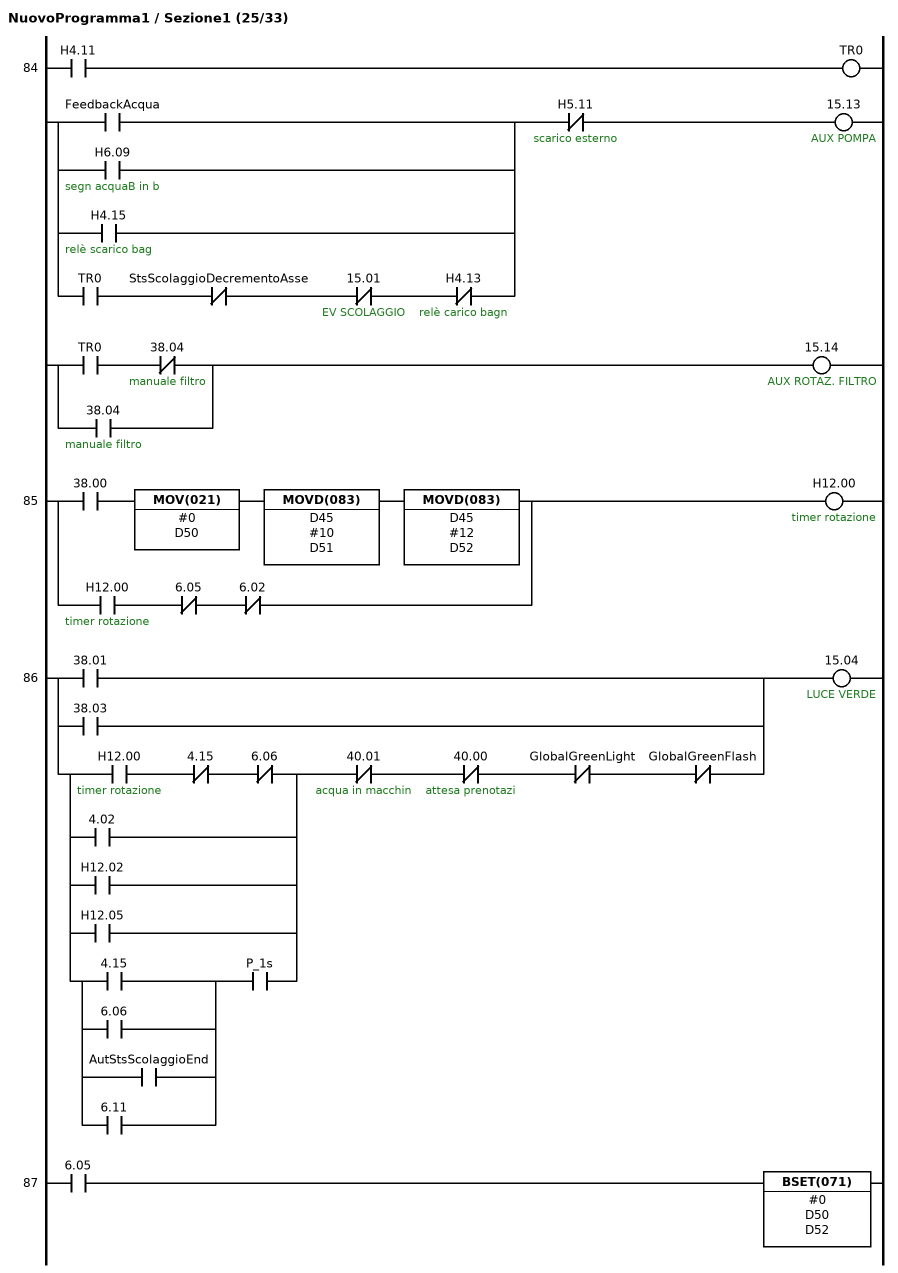
; [picture p24: NuovoProgramma1 / Sezione1, rungs 84-87]
; rung 84
LD FeedbackAcqua
OR H6.09  ; segn acquaB in b
OR H4.15  ; relè scarico bag
LD H4.11
OUT TR0
ANDNOT StsScolaggioDecrementoAsse
ANDNOT 15.01  ; EV SCOLAGGIO
ANDNOT H4.13  ; relè carico bagn
ORLD
ANDNOT H5.11  ; scarico esterno
OUT 15.13  ; AUX POMPA
LD TR0
ANDNOT 38.04  ; manuale filtro
OR 38.04  ; manuale filtro
OUT 15.14  ; AUX ROTAZ. FILTRO
; rung 85
LD 38.00
MOV(021) #0 D50
MOVD(083) D45 #10 D51
MOVD(083) D45 #12 D52
LD H12.00  ; timer rotazione
ANDNOT 6.05
ANDNOT 6.02
ORLD
OUT H12.00  ; timer rotazione
; rung 86
LD 38.01
OR 38.03
LD H12.00  ; timer rotazione
ANDNOT 4.15
ANDNOT 6.06
OR 4.02
OR H12.02
OR H12.05
LD 4.15
OR 6.06
OR AutStsScolaggioEnd
OR 6.11
AND P_1s
ORLD
ANDNOT 40.01  ; acqua in macchin
ANDNOT 40.00  ; attesa prenotazi
ANDNOT GlobalGreenLight
ANDNOT GlobalGreenFlash
ORLD
OUT 15.04  ; LUCE VERDE
; rung 87
LD 6.05
BSET(071) #0 D50 D52

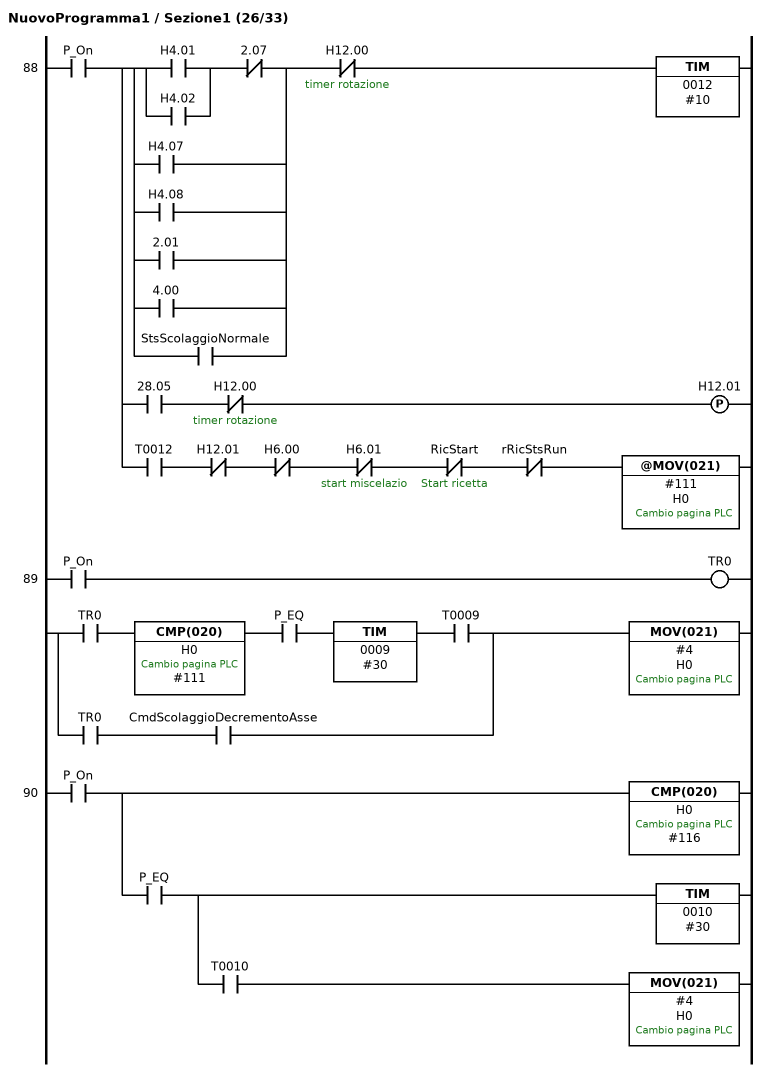
; rung 88
LD P_On
OUT TR0
LD H4.01
OR H4.02
ANDNOT 2.07
OR H4.07
OR H4.08
OR 2.01
OR 4.00
OR StsScolaggioNormale
ANDLD
ANDNOT H12.00  ; timer rotazione
TIM 0012 #10
LD TR0
AND 28.05
ANDNOT H12.00  ; timer rotazione
DIFU(013) H12.01
LD TR0
AND T0012
ANDNOT H12.01
ANDNOT H6.00
ANDNOT H6.01  ; start miscelazio
ANDNOT RicStart  ; Start ricetta
ANDNOT rRicStsRun
@MOV(021) #111 H0  ; Cambio pagina PLC
; rung 89
LD P_On
OUT TR0
CMP(020) H0 #111  ; Cambio pagina PLC
AND P_EQ
TIM 0009 #30
AND T0009
LD TR0
AND CmdScolaggioDecrementoAsse
ORLD
MOV(021) #4 H0  ; Cambio pagina PLC
; rung 90
LD P_On
CMP(020) H0 #116  ; Cambio pagina PLC
AND P_EQ
TIM 0010 #30
AND T0010
MOV(021) #4 H0  ; Cambio pagina PLC

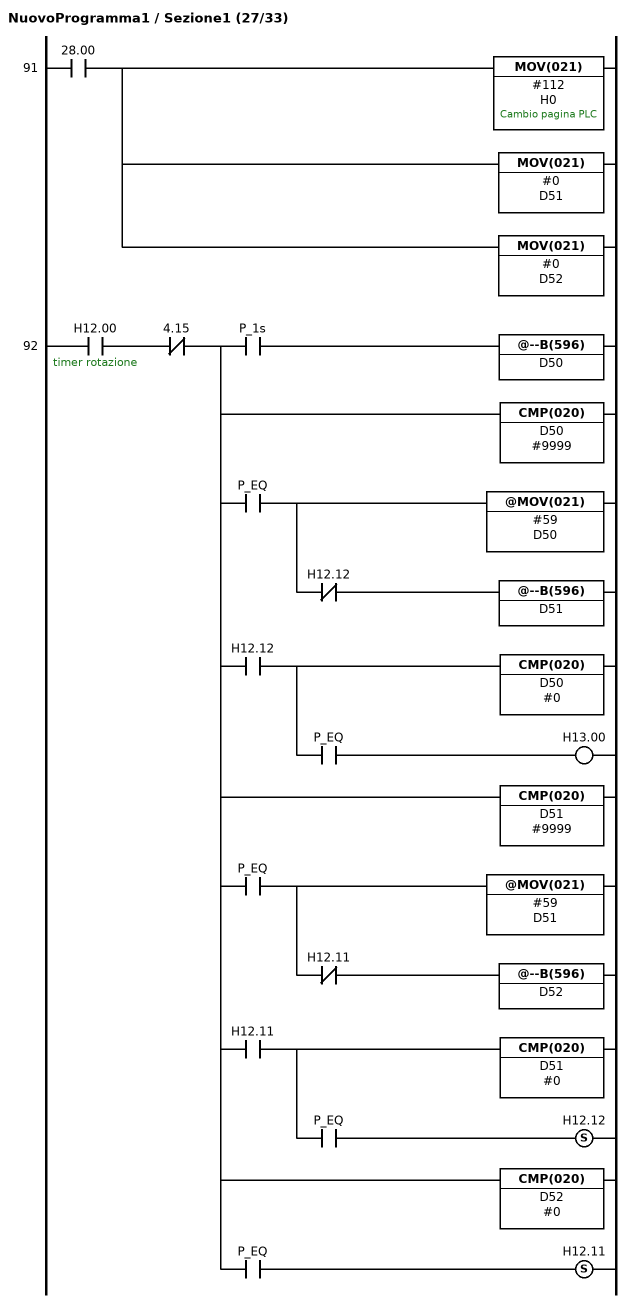
; rung 91
LD 28.00
MOV(021) #112 H0  ; Cambio pagina PLC
MOV(021) #0 D51
MOV(021) #0 D52
; rung 92
LD H12.00  ; timer rotazione
ANDNOT 4.15
OUT TR0
AND P_1s
@--B(596) D50
LD TR0
CMP(020) D50 #9999
AND P_EQ
@MOV(021) #59 D50
ANDNOT H12.12
@--B(596) D51
LD TR0
AND H12.12
CMP(020) D50 #0
AND P_EQ
OUT H13.00
LD TR0
CMP(020) D51 #9999
AND P_EQ
@MOV(021) #59 D51
ANDNOT H12.11
@--B(596) D52
LD TR0
AND H12.11
CMP(020) D51 #0
AND P_EQ
SET H12.12
LD TR0
CMP(020) D52 #0
AND P_EQ
SET H12.11

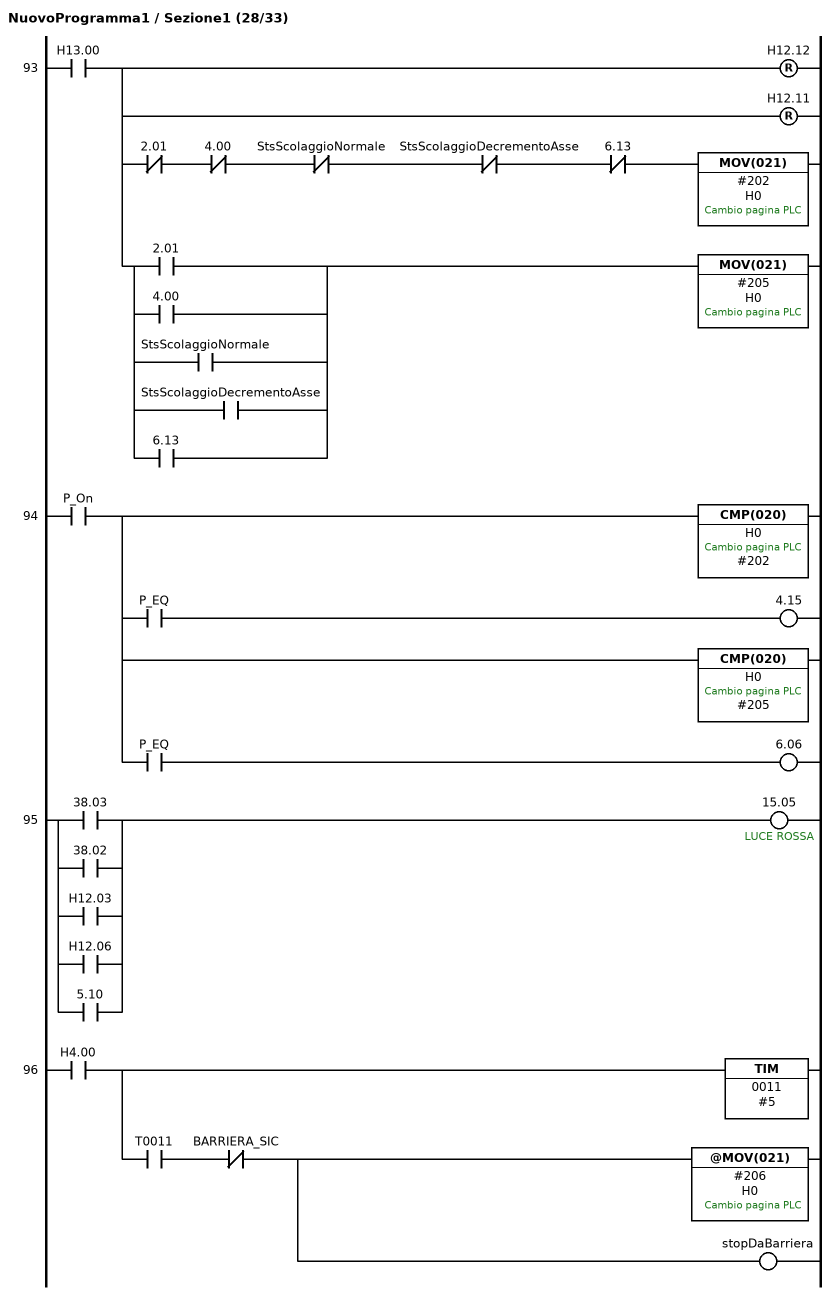
; rung 93
LD H13.00
OUT TR0
RSET H12.12
RSET H12.11
ANDNOT 2.01
ANDNOT 4.00
ANDNOT StsScolaggioNormale
ANDNOT StsScolaggioDecrementoAsse
ANDNOT 6.13
MOV(021) #202 H0  ; Cambio pagina PLC
LD TR0
LD 2.01
OR 4.00
OR StsScolaggioNormale
OR StsScolaggioDecrementoAsse
OR 6.13
ANDLD
MOV(021) #205 H0  ; Cambio pagina PLC
; rung 94
LD P_On
OUT TR0
CMP(020) H0 #202  ; Cambio pagina PLC
AND P_EQ
OUT 4.15
LD TR0
CMP(020) H0 #205  ; Cambio pagina PLC
AND P_EQ
OUT 6.06
; rung 95
LD 38.03
OR 38.02
OR H12.03
OR H12.06
OR 5.10
OUT 15.05  ; LUCE ROSSA
; rung 96
LD H4.00
TIM 0011 #5
AND T0011
ANDNOT BARRIERA_SIC
@MOV(021) #206 H0  ; Cambio pagina PLC
OUT stopDaBarriera

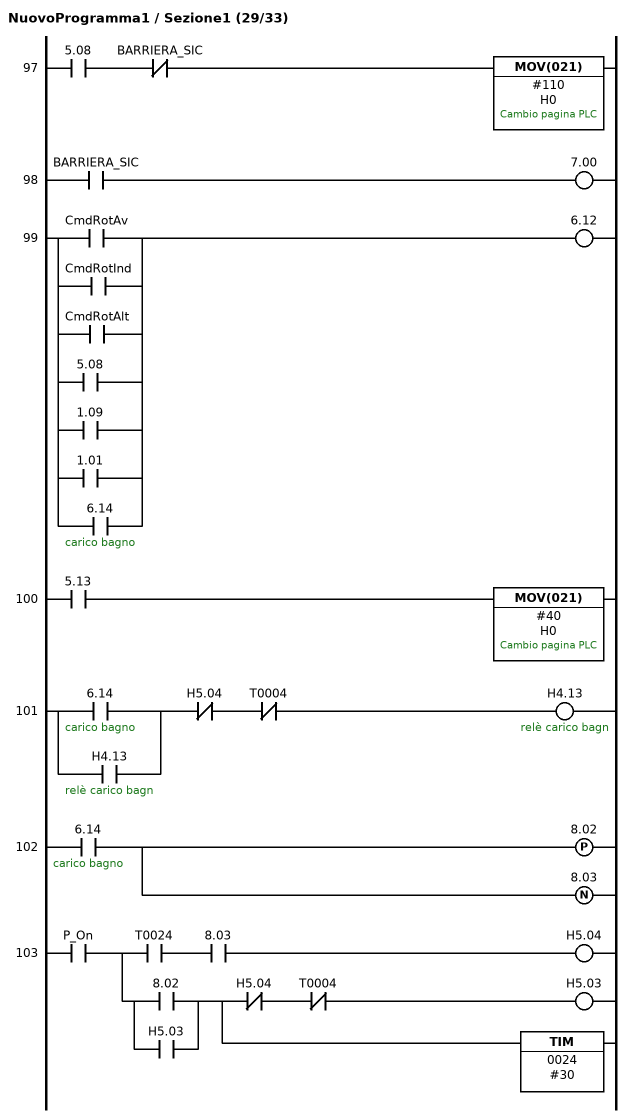
; rung 97
LD 5.08
ANDNOT BARRIERA_SIC
MOV(021) #110 H0  ; Cambio pagina PLC
; rung 98
LD BARRIERA_SIC
OUT 7.00
; rung 99
LD CmdRotAv
OR CmdRotInd
OR CmdRotAlt
OR 5.08
OR 1.09
OR 1.01
OR 6.14  ; carico bagno
OUT 6.12
; rung 100
LD 5.13
MOV(021) #40 H0  ; Cambio pagina PLC
; rung 101
LD 6.14  ; carico bagno
OR H4.13  ; relè carico bagn
ANDNOT H5.04
ANDNOT T0004
OUT H4.13  ; relè carico bagn
; rung 102
LD 6.14  ; carico bagno
DIFU(013) 8.02
DIFD(014) 8.03
; rung 103
LD P_On
OUT TR0
AND T0024
AND 8.03
OUT H5.04
LD TR0
LD 8.02
OR H5.03
ANDLD
OUT TR0
ANDNOT H5.04
ANDNOT T0004
OUT H5.03
LD TR0
TIM 0024 #30

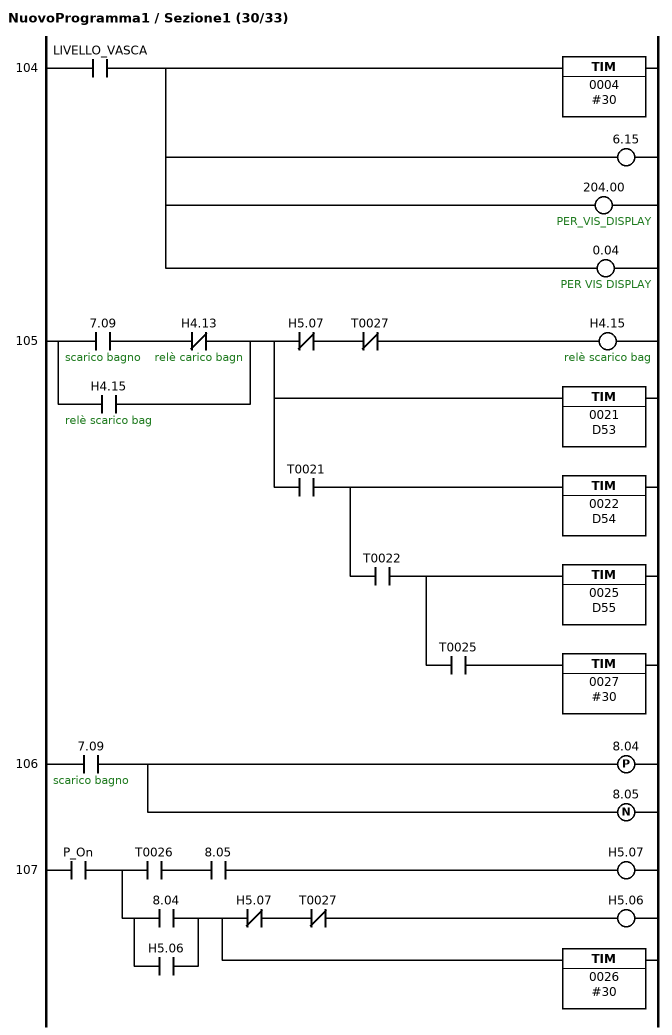
; rung 104
LD LIVELLO_VASCA
TIM 0004 #30
OUT 6.15
OUT 204.00  ; PER_VIS_DISPLAY
OUT 0.04  ; PER VIS DISPLAY
; rung 105
LD 7.09  ; scarico bagno
ANDNOT H4.13  ; relè carico bagn
OR H4.15  ; relè scarico bag
OUT TR0
ANDNOT H5.07
ANDNOT T0027
OUT H4.15  ; relè scarico bag
LD TR0
TIM 0021 D53
AND T0021
TIM 0022 D54
AND T0022
TIM 0025 D55
AND T0025
TIM 0027 #30
; rung 106
LD 7.09  ; scarico bagno
DIFU(013) 8.04
DIFD(014) 8.05
; rung 107
LD P_On
OUT TR0
AND T0026
AND 8.05
OUT H5.07
LD TR0
LD 8.04
OR H5.06
ANDLD
OUT TR0
ANDNOT H5.07
ANDNOT T0027
OUT H5.06
LD TR0
TIM 0026 #30

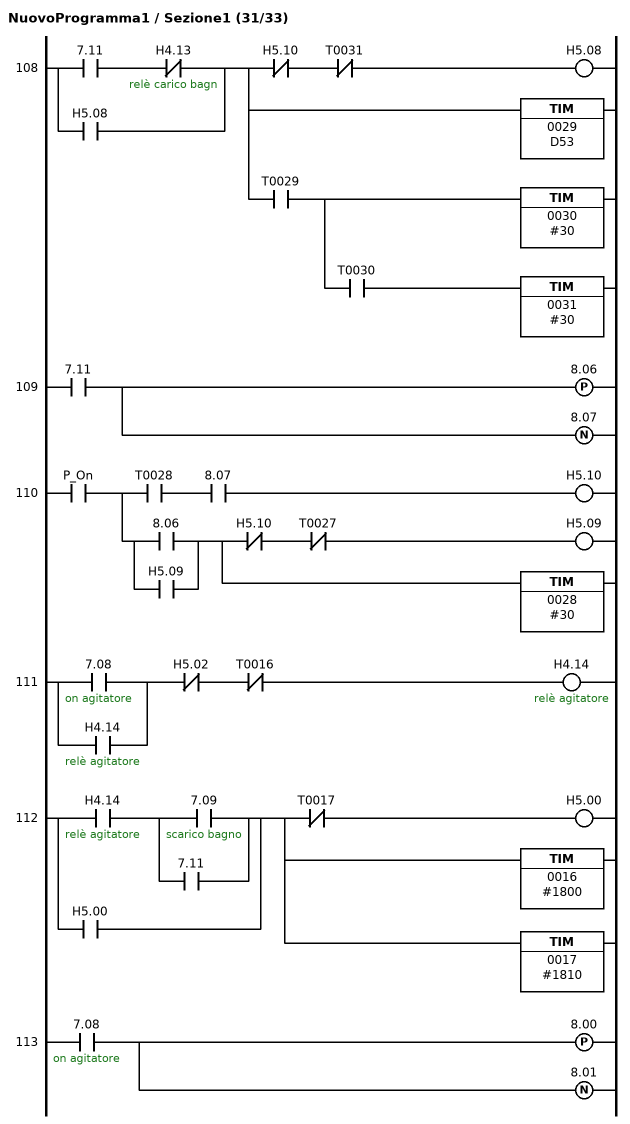
; rung 108
LD 7.11
ANDNOT H4.13  ; relè carico bagn
OR H5.08
OUT TR0
ANDNOT H5.10
ANDNOT T0031
OUT H5.08
LD TR0
TIM 0029 D53
AND T0029
TIM 0030 #30
AND T0030
TIM 0031 #30
; rung 109
LD 7.11
DIFU(013) 8.06
DIFD(014) 8.07
; rung 110
LD P_On
OUT TR0
AND T0028
AND 8.07
OUT H5.10
LD TR0
LD 8.06
OR H5.09
ANDLD
OUT TR0
ANDNOT H5.10
ANDNOT T0027
OUT H5.09
LD TR0
TIM 0028 #30
; rung 111
LD 7.08  ; on agitatore
OR H4.14  ; relè agitatore
ANDNOT H5.02
ANDNOT T0016
OUT H4.14  ; relè agitatore
; rung 112
LD H4.14  ; relè agitatore
LD 7.09  ; scarico bagno
OR 7.11
ANDLD
OR H5.00
OUT TR0
ANDNOT T0017
OUT H5.00
LD TR0
TIM 0016 #1800
TIM 0017 #1810
; rung 113
LD 7.08  ; on agitatore
DIFU(013) 8.00
DIFD(014) 8.01

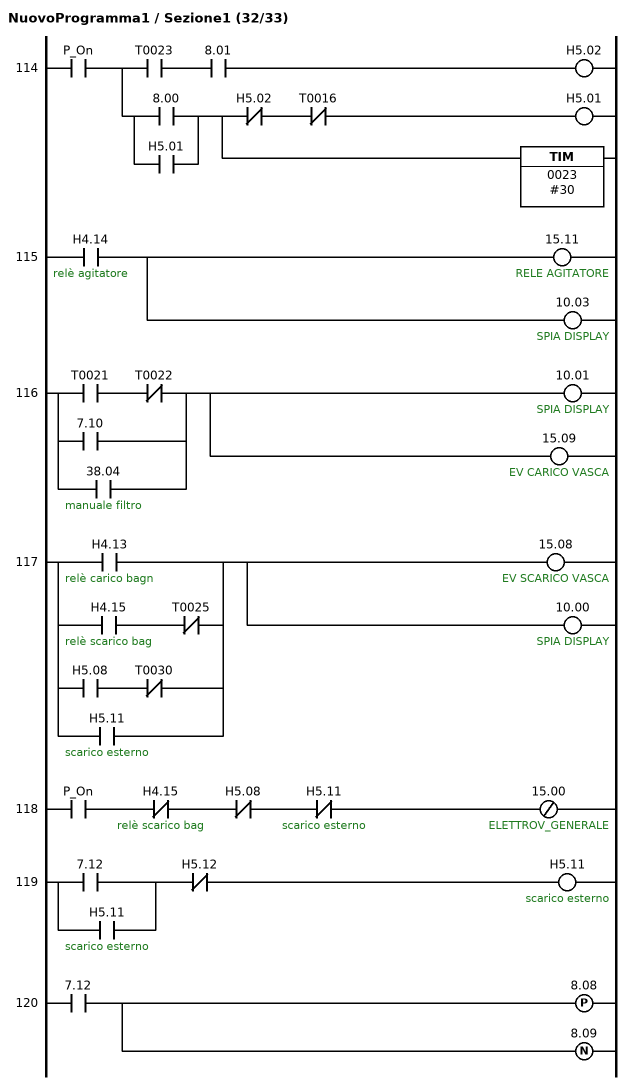
; rung 114
LD P_On
OUT TR0
AND T0023
AND 8.01
OUT H5.02
LD TR0
LD 8.00
OR H5.01
ANDLD
OUT TR0
ANDNOT H5.02
ANDNOT T0016
OUT H5.01
LD TR0
TIM 0023 #30
; rung 115
LD H4.14  ; relè agitatore
OUT 15.11  ; RELE AGITATORE
OUT 10.03  ; SPIA DISPLAY
; rung 116
LD T0021
ANDNOT T0022
OR 7.10
OR 38.04  ; manuale filtro
OUT 10.01  ; SPIA DISPLAY
OUT 15.09  ; EV CARICO VASCA
; rung 117
LD H4.13  ; relè carico bagn
LD H4.15  ; relè scarico bag
ANDNOT T0025
ORLD
LD H5.08
ANDNOT T0030
ORLD
OR H5.11  ; scarico esterno
OUT 15.08  ; EV SCARICO VASCA
OUT 10.00  ; SPIA DISPLAY
; rung 118
LD P_On
ANDNOT H4.15  ; relè scarico bag
ANDNOT H5.08
ANDNOT H5.11  ; scarico esterno
OUTNOT 15.00  ; ELETTROV_GENERALE
; rung 119
LD 7.12
OR H5.11  ; scarico esterno
ANDNOT H5.12
OUT H5.11  ; scarico esterno
; rung 120
LD 7.12
DIFU(013) 8.08
DIFD(014) 8.09

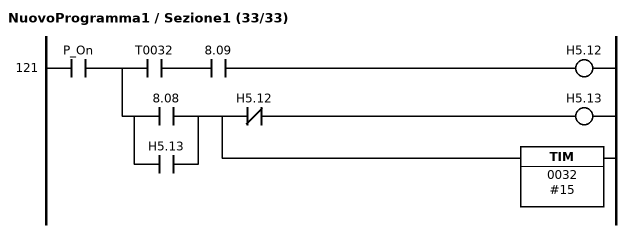
; rung 121
LD P_On
OUT TR0
AND T0032
AND 8.09
OUT H5.12
LD TR0
LD 8.08
OR H5.13
ANDLD
OUT TR0
ANDNOT H5.12
OUT H5.13
LD TR0
TIM 0032 #15

### Section Sezione2

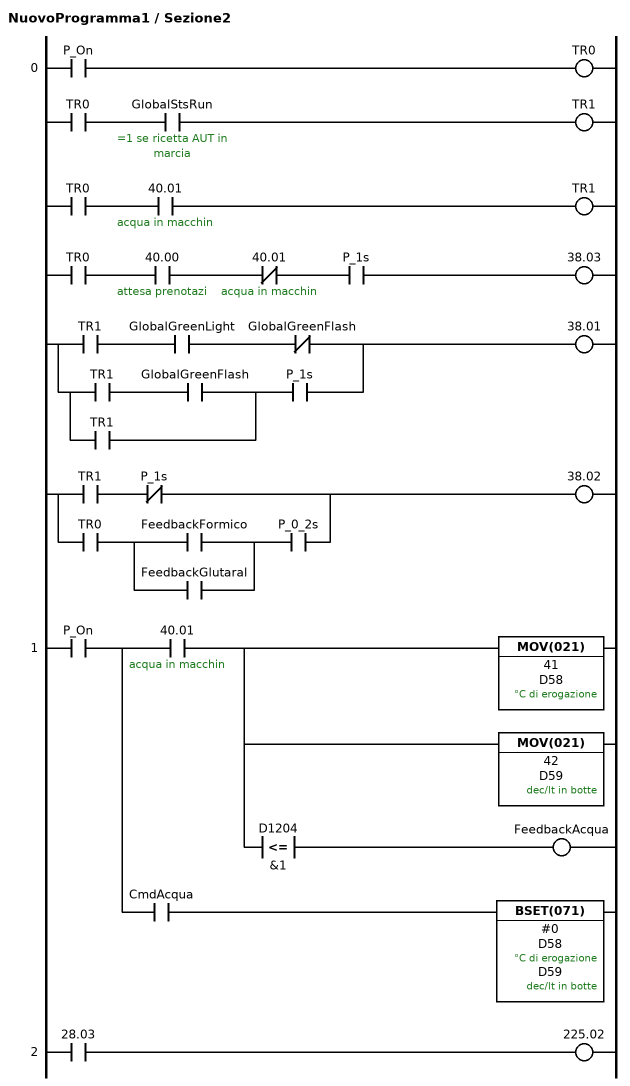
; rung 0
LD P_On
OUT TR0
AND 40.00  ; attesa prenotazi
ANDNOT 40.01  ; acqua in macchin
AND P_1s
OUT 38.03
LD TR0
AND GlobalStsRun  ; =1 se ricetta AUT in marcia
OUT TR1
AND GlobalGreenLight
ANDNOT GlobalGreenFlash
LD TR1
AND GlobalGreenFlash
LD TR0
AND 40.01  ; acqua in macchin
OUT TR1
ORLD
AND P_1s
ORLD
OUT 38.01
LD TR1
ANDNOT P_1s
LD TR0
LD FeedbackFormico
OR FeedbackGlutaral
ANDLD
AND P_0_2s
ORLD
OUT 38.02
; rung 1
LD P_On
OUT TR0
AND 40.01  ; acqua in macchin
MOV(021) 41 D58  ; °C di erogazione
MOV(021) 42 D59  ; dec/lt in botte
AND<=(315) D1204 &1
OUT FeedbackAcqua
LD TR0
AND CmdAcqua
BSET(071) #0 D58 D59  ; °C di erogazione, dec/lt in botte
; rung 2
LD 28.03
OUT 225.02

### Section Sezione3

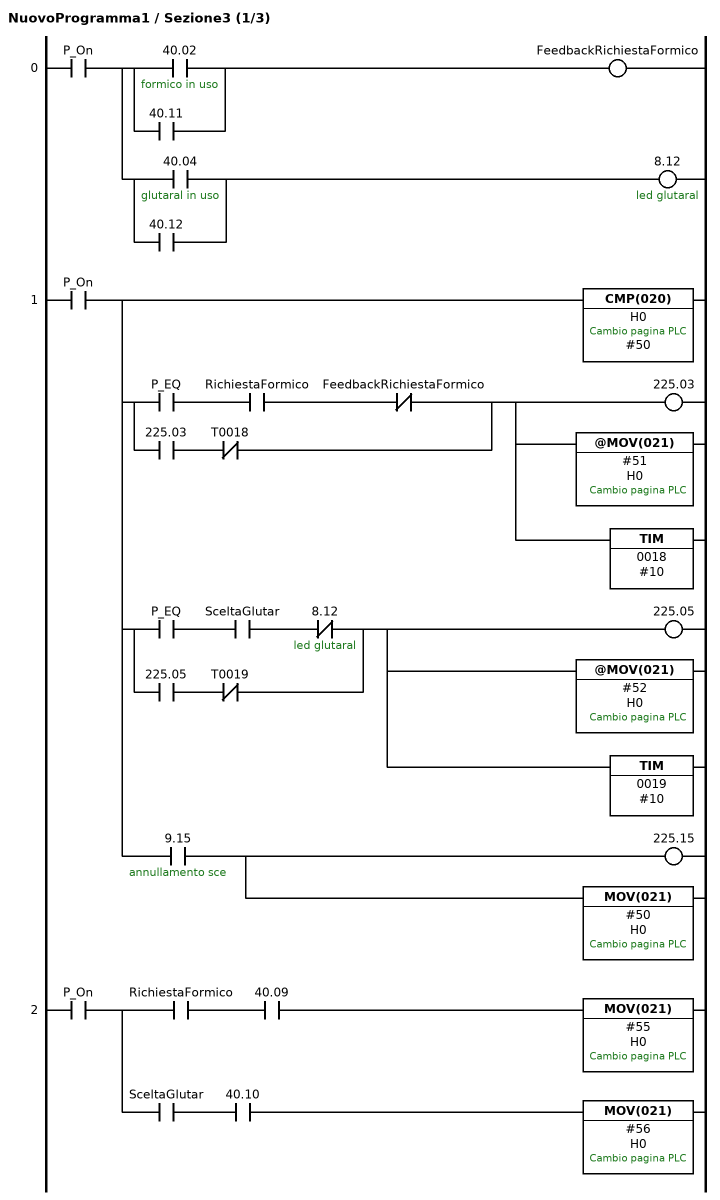
; rung 0
LD P_On
OUT TR0
LD 40.02  ; formico in uso
OR 40.11
ANDLD
OUT FeedbackRichiestaFormico
LD TR0
LD 40.04  ; glutaral in uso
OR 40.12
ANDLD
OUT 8.12  ; led glutaral
; rung 1
LD P_On
OUT TR0
CMP(020) H0 #50  ; Cambio pagina PLC
LD P_EQ
AND RichiestaFormico
ANDNOT FeedbackRichiestaFormico
LD 225.03
ANDNOT T0018
ORLD
ANDLD
OUT 225.03
@MOV(021) #51 H0  ; Cambio pagina PLC
TIM 0018 #10
LD TR0
LD P_EQ
AND SceltaGlutar
ANDNOT 8.12  ; led glutaral
LD 225.05
ANDNOT T0019
ORLD
ANDLD
OUT 225.05
@MOV(021) #52 H0  ; Cambio pagina PLC
TIM 0019 #10
LD TR0
AND 9.15  ; annullamento sce
OUT 225.15
MOV(021) #50 H0  ; Cambio pagina PLC
; rung 2
LD P_On
OUT TR0
AND RichiestaFormico
AND 40.09
MOV(021) #55 H0  ; Cambio pagina PLC
LD TR0
AND SceltaGlutar
AND 40.10
MOV(021) #56 H0  ; Cambio pagina PLC

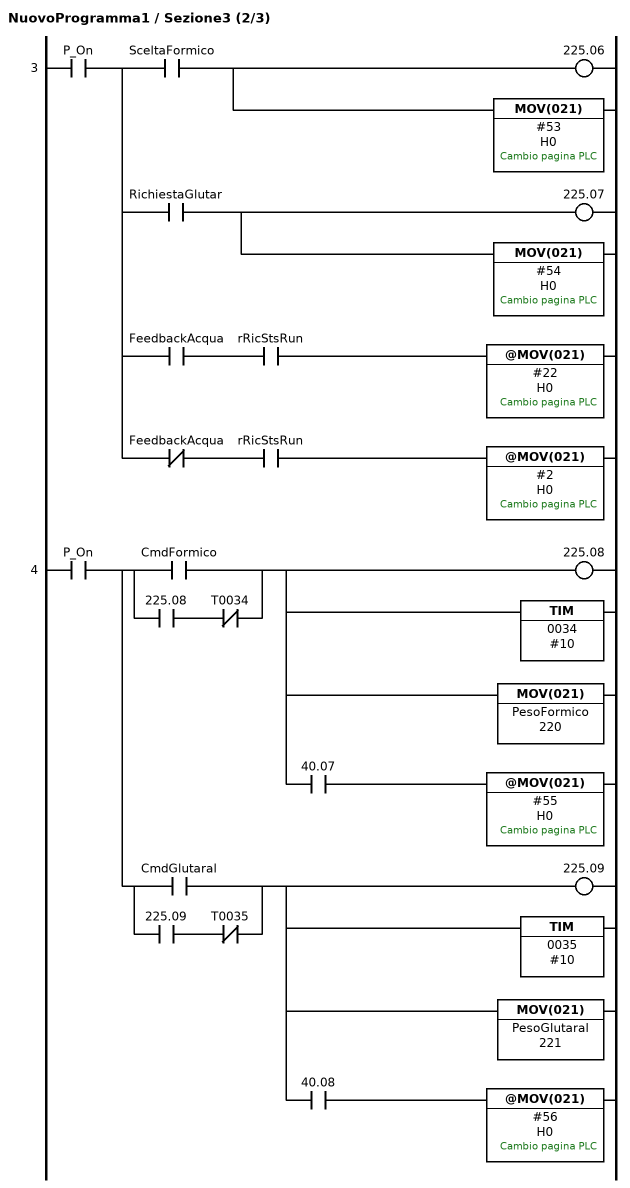
; rung 3
LD P_On
OUT TR0
AND SceltaFormico
OUT 225.06
MOV(021) #53 H0  ; Cambio pagina PLC
LD TR0
AND RichiestaGlutar
OUT 225.07
MOV(021) #54 H0  ; Cambio pagina PLC
LD TR0
AND FeedbackAcqua
AND rRicStsRun
@MOV(021) #22 H0  ; Cambio pagina PLC
LD TR0
ANDNOT FeedbackAcqua
AND rRicStsRun
@MOV(021) #2 H0  ; Cambio pagina PLC
; rung 4
LD P_On
OUT TR0
LD CmdFormico
LD 225.08
ANDNOT T0034
ORLD
ANDLD
OUT 225.08
TIM 0034 #10
MOV(021) PesoFormico 220
AND 40.07
@MOV(021) #55 H0  ; Cambio pagina PLC
LD TR0
LD CmdGlutaral
LD 225.09
ANDNOT T0035
ORLD
ANDLD
OUT 225.09
TIM 0035 #10
MOV(021) PesoGlutaral 221
AND 40.08
@MOV(021) #56 H0  ; Cambio pagina PLC

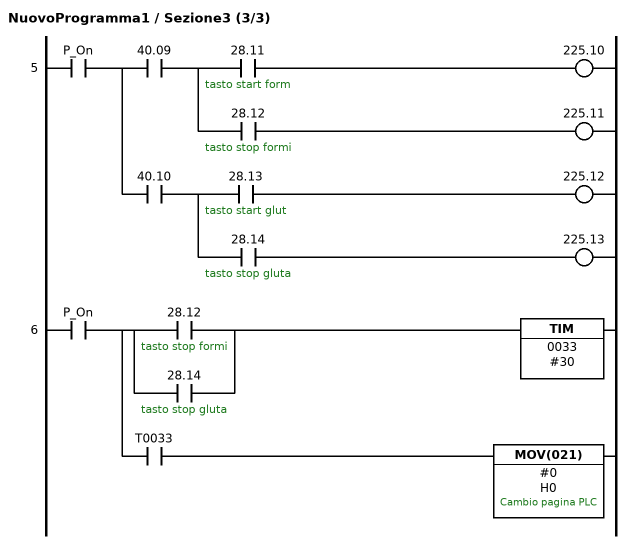
; rung 5
LD P_On
OUT TR0
AND 40.09
OUT TR1
AND 28.11  ; tasto start form
OUT 225.10
LD TR1
AND 28.12  ; tasto stop formi
OUT 225.11
LD TR0
AND 40.10
OUT TR0
AND 28.13  ; tasto start glut
OUT 225.12
LD TR0
AND 28.14  ; tasto stop gluta
OUT 225.13
; rung 6
LD P_On
OUT TR0
LD 28.12  ; tasto stop formi
OR 28.14  ; tasto stop gluta
ANDLD
TIM 0033 #30
LD TR0
AND T0033
MOV(021) #0 H0  ; Cambio pagina PLC
; rung 7
END(001)

## Program TaskRicette (cyclic task 1)

### Section CambioPagina

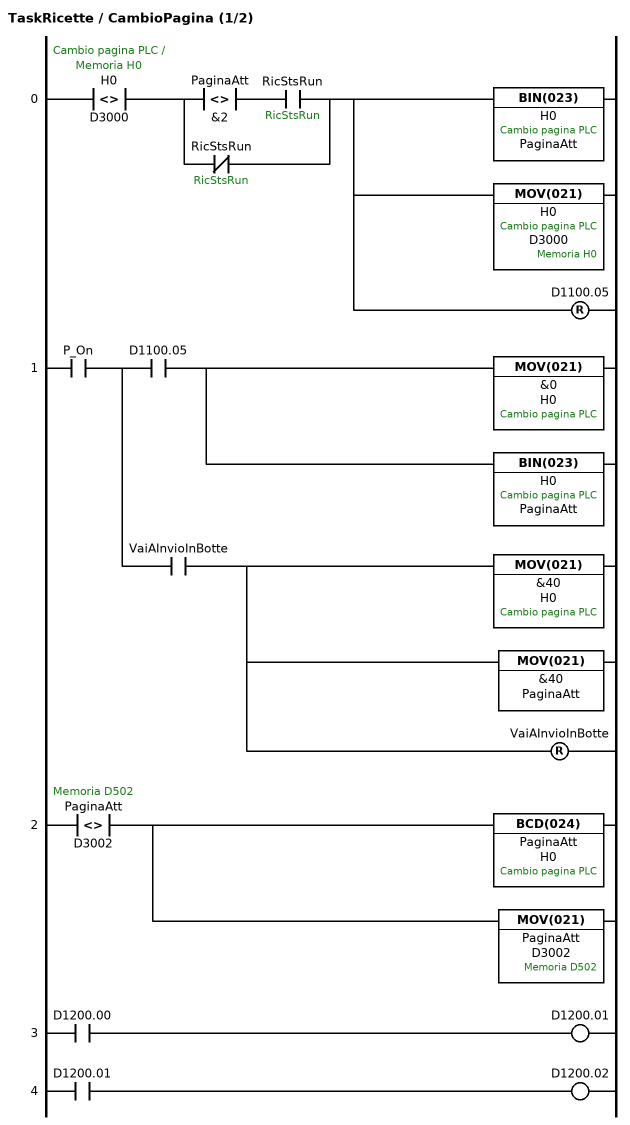
; rung 0
LD<>(305) H0 D3000  ; Cambio pagina PLC, Memoria H0
LD<>(305) PaginaAtt &2
AND RicStsRun  ; RicStsRun
ORNOT RicStsRun  ; RicStsRun
ANDLD
BIN(023) H0 PaginaAtt  ; Cambio pagina PLC
MOV(021) H0 D3000  ; Cambio pagina PLC, Memoria H0
RSET D1100.05
; rung 1
LD P_On
OUT TR0
AND D1100.05
MOV(021) &0 H0  ; Cambio pagina PLC
BIN(023) H0 PaginaAtt  ; Cambio pagina PLC
LD TR0
AND VaiAInvioInBotte
MOV(021) &40 H0  ; Cambio pagina PLC
MOV(021) &40 PaginaAtt
RSET VaiAInvioInBotte
; rung 2
LD<>(305) PaginaAtt D3002  ; Memoria D502
BCD(024) PaginaAtt H0  ; Cambio pagina PLC
MOV(021) PaginaAtt D3002  ; Memoria D502
; rung 3
LD D1200.00
OUT D1200.01
; rung 4
LD D1200.01
OUT D1200.02

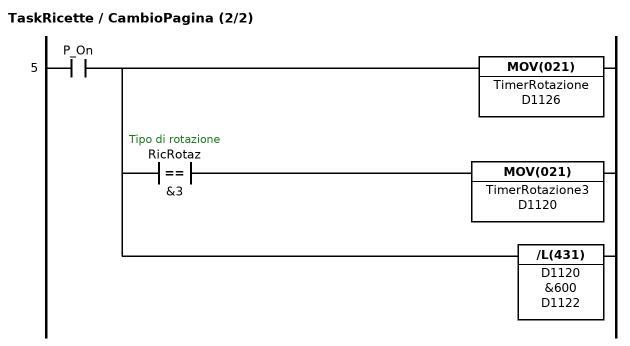
; rung 5
LD P_On
OUT TR0
MOV(021) TimerRotazione D1126
AND=(300) RicRotaz &3  ; Tipo di rotazione
MOV(021) TimerRotazione3 D1120
LD TR0
/L(431) D1120 &600 D1122

### Section Puntatori

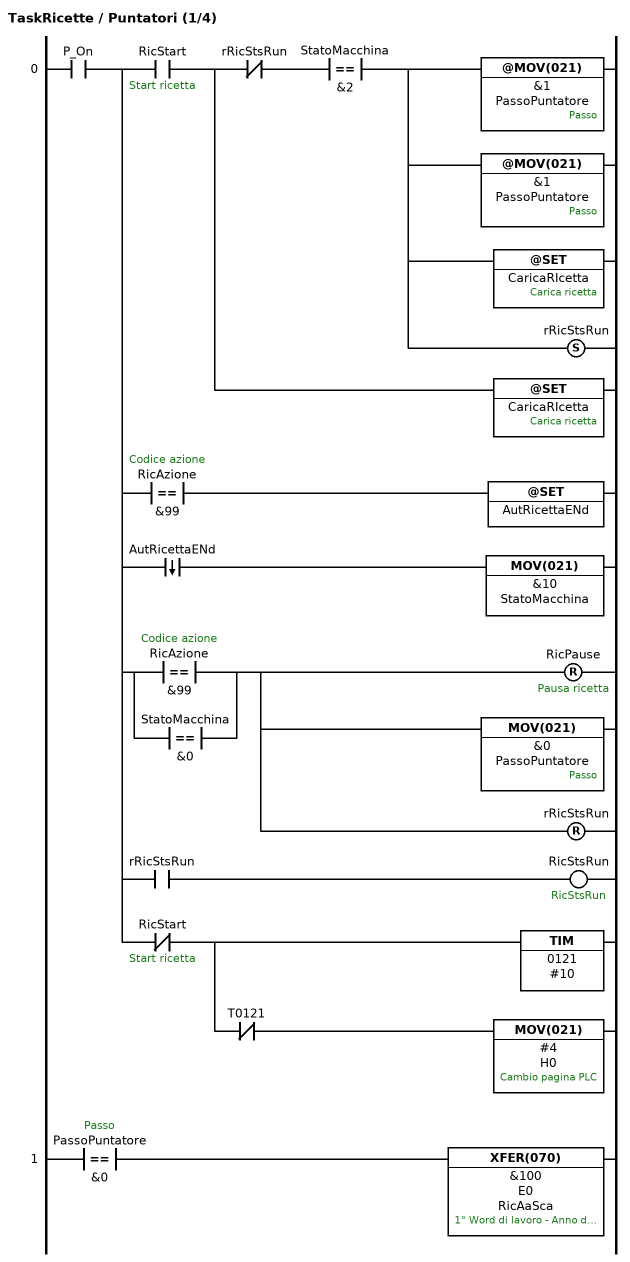
; rung 0
LD P_On
OUT TR0
AND RicStart  ; Start ricetta
OUT TR1
ANDNOT rRicStsRun
AND=(300) StatoMacchina &2
@MOV(021) &1 PassoPuntatore  ; Passo
@MOV(021) &1 PassoPuntatore  ; Passo
@SET CaricaRIcetta  ; Carica ricetta
SET rRicStsRun
LD TR1
@SET CaricaRIcetta  ; Carica ricetta
LD TR0
AND=(300) RicAzione &99  ; Codice azione
@SET AutRicettaENd
LD TR0
%AND AutRicettaENd
MOV(021) &10 StatoMacchina
LD TR0
LD=(300) RicAzione &99  ; Codice azione
OR=(300) StatoMacchina &0
ANDLD
RSET RicPause  ; Pausa ricetta
MOV(021) &0 PassoPuntatore  ; Passo
RSET rRicStsRun
LD TR0
AND rRicStsRun
OUT RicStsRun  ; RicStsRun
LD TR0
ANDNOT RicStart  ; Start ricetta
TIM 0121 #10
ANDNOT T0121
MOV(021) #4 H0  ; Cambio pagina PLC
; rung 1
LD=(300) PassoPuntatore &0  ; Passo
XFER(070) &100 E0 RicAaSca  ; 1° Word di lavoro - Anno di produzione

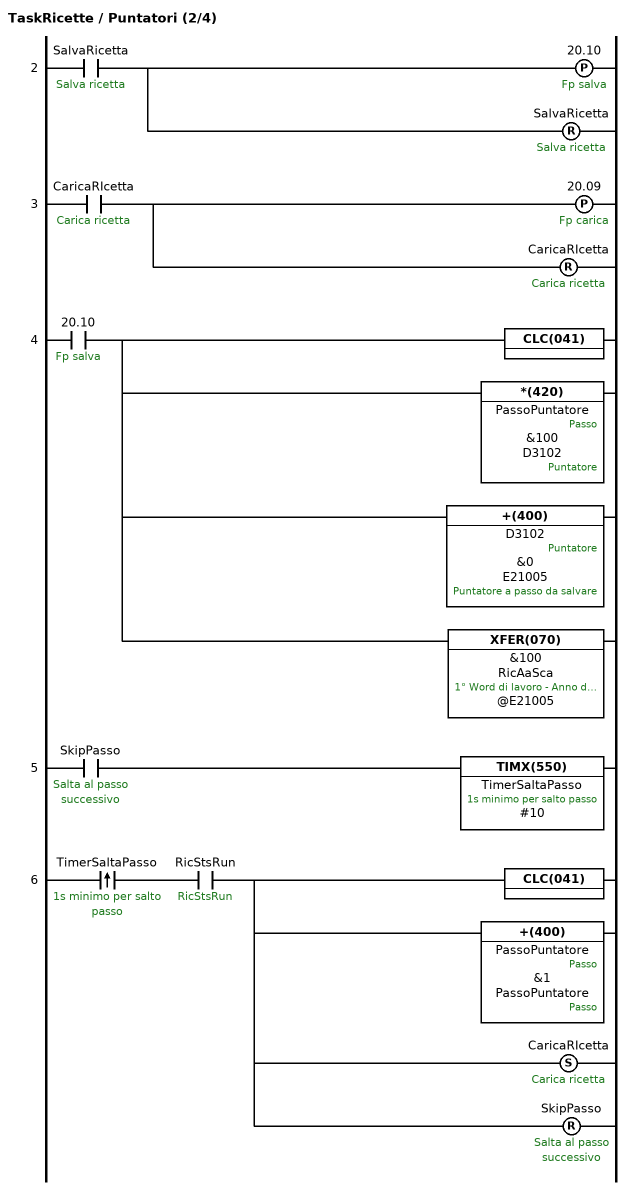
; rung 2
LD SalvaRicetta  ; Salva ricetta
DIFU(013) 20.10  ; Fp salva
RSET SalvaRicetta  ; Salva ricetta
; rung 3
LD CaricaRIcetta  ; Carica ricetta
DIFU(013) 20.09  ; Fp carica
RSET CaricaRIcetta  ; Carica ricetta
; rung 4
LD 20.10  ; Fp salva
CLC(041)
*(420) PassoPuntatore &100 D3102  ; Passo, Puntatore
+(400) D3102 &0 E21005  ; Puntatore, Puntatore a passo da salvare
XFER(070) &100 RicAaSca @E21005  ; 1° Word di lavoro - Anno di produzione
; rung 5
LD SkipPasso  ; Salta al passo successivo
TIMX(550) TimerSaltaPasso #10  ; 1s minimo per salto passo
; rung 6
@LD TimerSaltaPasso  ; 1s minimo per salto passo
AND RicStsRun  ; RicStsRun
CLC(041)
+(400) PassoPuntatore &1 PassoPuntatore  ; Passo
SET CaricaRIcetta  ; Carica ricetta
RSET SkipPasso  ; Salta al passo successivo

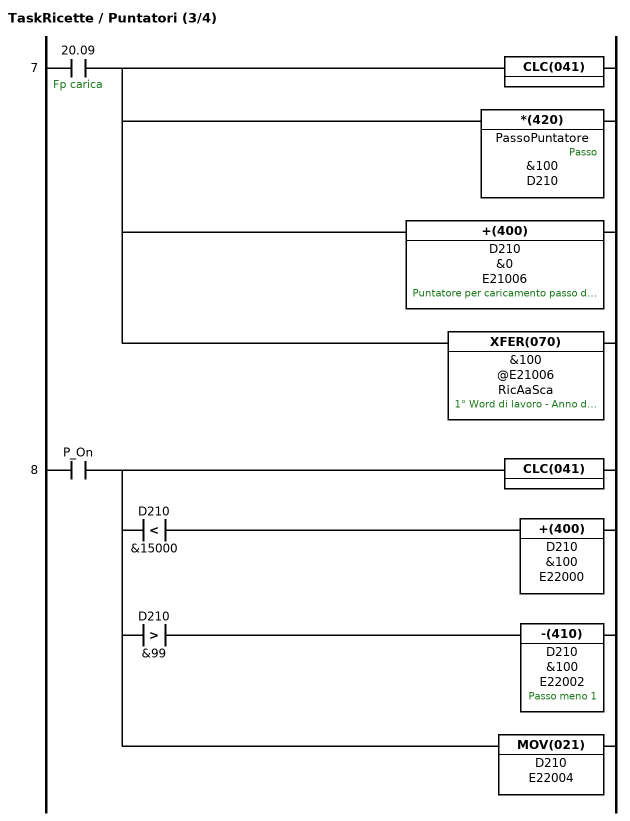
; rung 7
LD 20.09  ; Fp carica
CLC(041)
*(420) PassoPuntatore &100 D210  ; Passo
+(400) D210 &0 E21006  ; Puntatore per caricamento passo da DB a lavoro
XFER(070) &100 @E21006 RicAaSca  ; 1° Word di lavoro - Anno di produzione
; rung 8
LD P_On
OUT TR0
CLC(041)
AND<(310) D210 &15000
+(400) D210 &100 E22000
LD TR0
AND>(320) D210 &99
-(410) D210 &100 E22002  ; Passo meno 1
LD TR0
MOV(021) D210 E22004

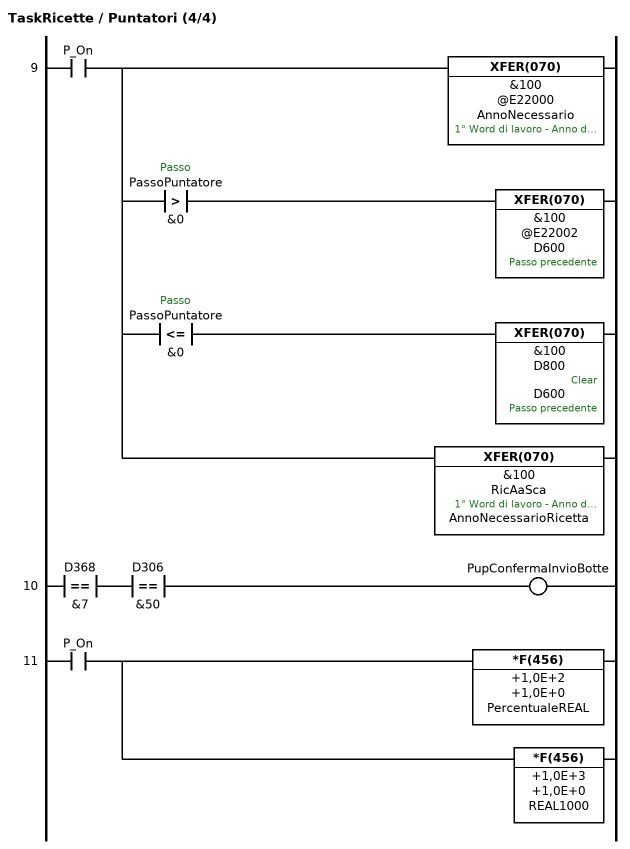
; rung 9
LD P_On
OUT TR0
XFER(070) &100 @E22000 AnnoNecessario  ; 1° Word di lavoro - Anno di produzione
AND>(320) PassoPuntatore &0  ; Passo
XFER(070) &100 @E22002 D600  ; Passo precedente
LD TR0
AND<=(315) PassoPuntatore &0  ; Passo
XFER(070) &100 D800 D600  ; Clear, Passo precedente
LD TR0
XFER(070) &100 RicAaSca AnnoNecessarioRicetta  ; 1° Word di lavoro - Anno di produzione
; rung 10
LD=(300) D368 &7
AND=(300) D306 &50
OUT PupConfermaInvioBotte
; rung 11
LD P_On
*F(456) +1,0E+2 +1,0E+0 PercentualeREAL
*F(456) +1,0E+3 +1,0E+0 REAL1000

### Section StatoRicetta

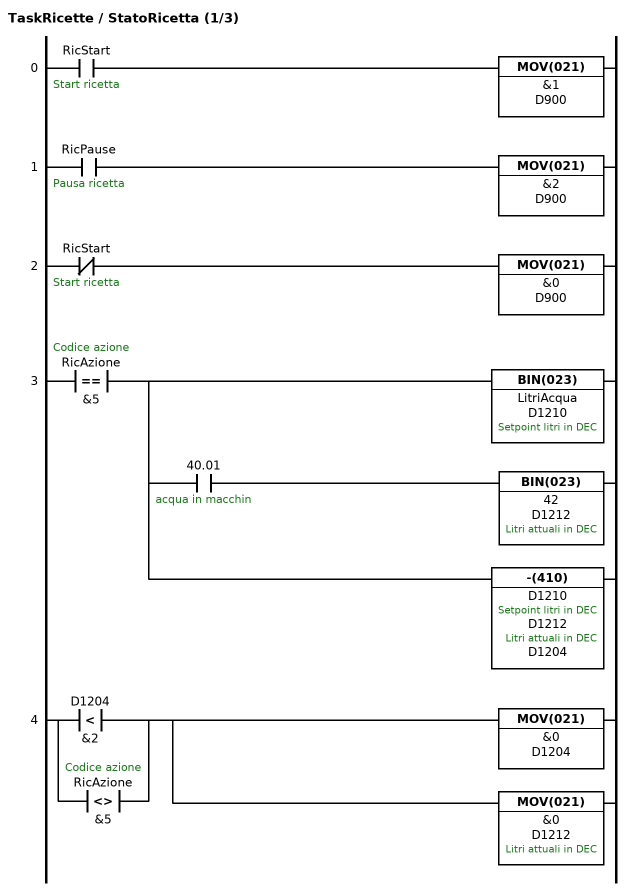
; rung 0
LD RicStart  ; Start ricetta
MOV(021) &1 D900
; rung 1
LD RicPause  ; Pausa ricetta
MOV(021) &2 D900
; rung 2
LDNOT RicStart  ; Start ricetta
MOV(021) &0 D900
; rung 3
LD=(300) RicAzione &5  ; Codice azione
OUT TR0
BIN(023) LitriAcqua D1210  ; Setpoint litri in DEC
AND 40.01  ; acqua in macchin
BIN(023) 42 D1212  ; Litri attuali in DEC
LD TR0
-(410) D1210 D1212 D1204  ; Setpoint litri in DEC, Litri attuali in DEC
; rung 4
LD<(310) D1204 &2
OR<>(305) RicAzione &5  ; Codice azione
MOV(021) &0 D1204
MOV(021) &0 D1212  ; Litri attuali in DEC

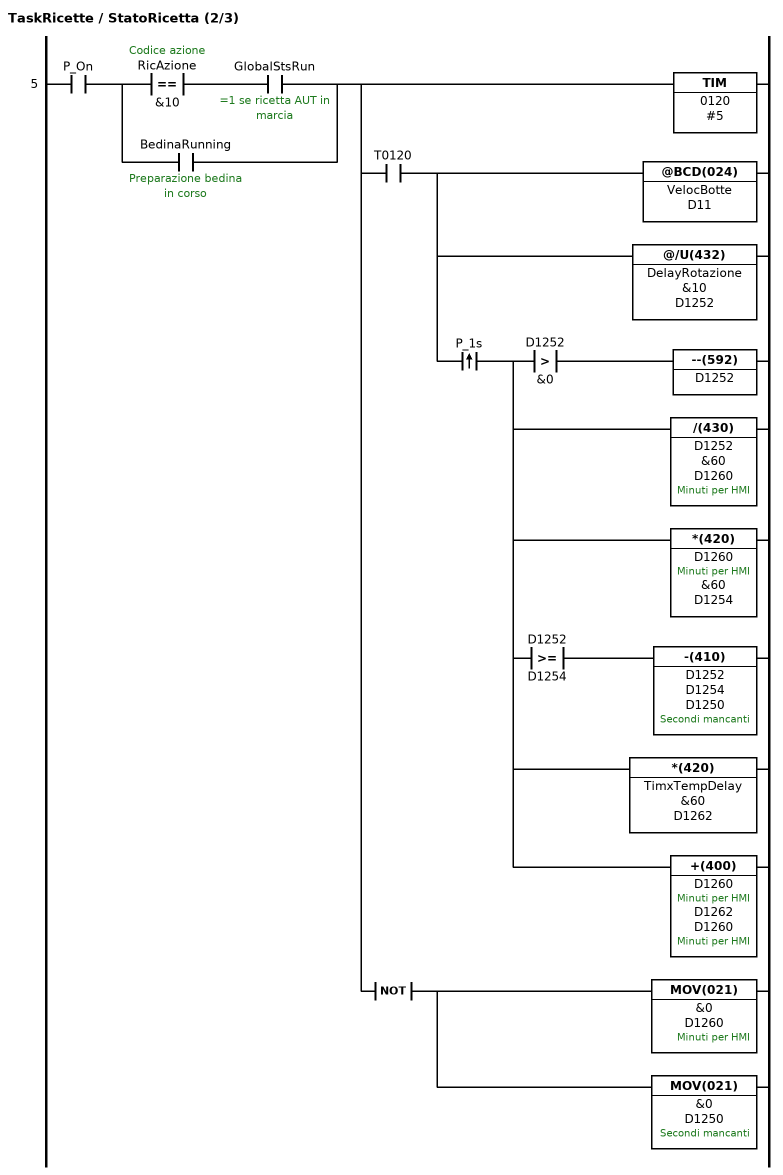
; rung 5
LD P_On
LD=(300) RicAzione &10  ; Codice azione
AND GlobalStsRun  ; =1 se ricetta AUT in marcia
OR BedinaRunning  ; Preparazione bedina in corso
ANDLD
OUT TR0
TIM 0120 #5
AND T0120
@BCD(024) VelocBotte D11
@/U(432) DelayRotazione &10 D1252
@AND P_1s
OUT TR1
AND>(320) D1252 &0
--(592) D1252
LD TR1
/(430) D1252 &60 D1260  ; Minuti per HMI
*(420) D1260 &60 D1254  ; Minuti per HMI
AND>=(325) D1252 D1254
-(410) D1252 D1254 D1250  ; Secondi mancanti
LD TR1
*(420) TimxTempDelay &60 D1262
+(400) D1260 D1262 D1260  ; Minuti per HMI
LD TR0
NOT(520)
MOV(021) &0 D1260  ; Minuti per HMI
MOV(021) &0 D1250  ; Secondi mancanti

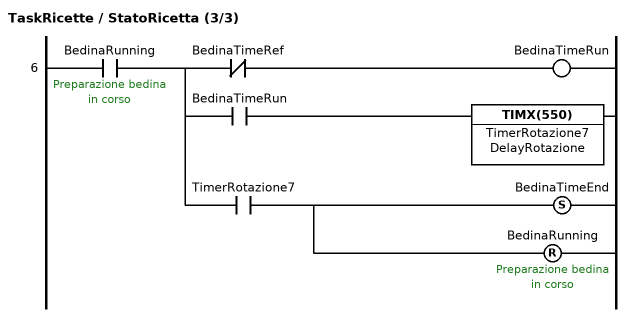
; rung 6
LD BedinaRunning  ; Preparazione bedina in corso
OUT TR0
ANDNOT BedinaTimeRef
OUT BedinaTimeRun
LD TR0
AND BedinaTimeRun
TIMX(550) TimerRotazione7 DelayRotazione
LD TR0
AND TimerRotazione7
SET BedinaTimeEnd
RSET BedinaRunning  ; Preparazione bedina in corso

### Section END

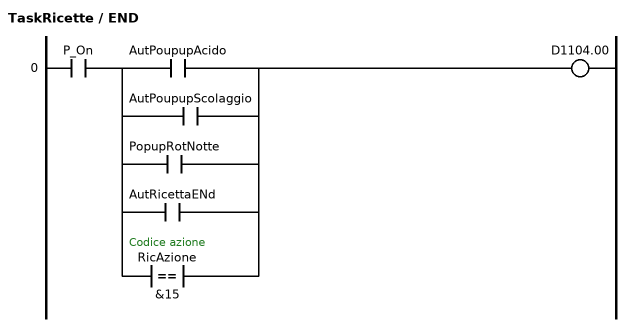
; rung 0
LD P_On
LD AutPoupupAcido
OR AutPoupupScolaggio
OR PopupRotNotte
OR AutRicettaENd
OR=(300) RicAzione &15  ; Codice azione
ANDLD
OUT D1104.00
; rung 1
END(001)

## Program CicliStep (cyclic task 2)
Local symbols
CmdRst D2000.00 BOOL
CmdStart D2000.01 BOOL
Index D2010 INT
MemRiga D2012 WORD
StepCiclo D2001.00 BOOL[15]
StsEnd D2000.02 BOOL
StsRun D2000.03 BOOL
TempAnnoNecessario D2016 DINT
i D2014 INT
 IF TimerSaltaPasso.CF = TRUE  AND MemTimSkip=FALSE THEN
	Index:= 1;
	CmdRotAv:= false;
	CmdRotInd:= false;
	CmdRotAlt:= false;
	CmdRotStop:= false;
	CmdRotNotte:= false;
	CmdAcqua:= false;
	CmdFormico:= false;
	CmdGlutaral:= false;
	CmdScolaggioDecrementoAsse:= false;
	CmdScolaggioNormale:= false;
	PopupMancatoScolaggio:= false;
	RichiestaLetturaBarcode:= false;
	AutCmdNotturno:= false;
	AutPoupupScolaggio:= false;

end_if;
MemTimSkip:= TimerSaltaPasso.CF;
 
 (*Stop Riga*)
IF NOT  RicStart then
	StsRun:= false;
	StsEnd:= true;
	Index:= 5;
END_IF;
 
 
 (* Reset ciclo e comandi vari *)
IF CmdRst = TRUE THEN
	StsRun:= false;
	CmdStart:= false;
	CmdRst := false;	
END_IF;
GlobalGreenFlash:= false;
GlobalGreenLight:= false;
LetturaPesoREAL:= DINT_TO_REAL(LetturaPesoDINT);
		LetturaPesoREAL:= LetturaPesoREAL/1000,0;
		TolleranzaInf:= PesoNecessarioRicetta-((PesoNecessarioRicetta*Tolleranza)/100,0);
	(*I comandi da temperatura sono SET, vengono resettati dopo 1s sennò non li prende usando il momentaneo*)
TIMX(CmdTemperaturaON=true,TimerPIDon,10);
TIMX(CmdTemperaturaOFF=true,TimerPIDoff,10);
IF TimerPIDon.CF=TRUE THEN
	CmdTemperaturaON:= false;
END_IF;
IF TimerPIDoff.CF=TRUE THEN
	CmdTemperaturaOFF:= false;
END_IF;
(*Salvataggio ID riga per cambio riga*)
IF RicRigNum<>MemRiga THEN
	CmdStart:= true;
END_IF;
MemRiga:= RicRigNum;

(* Start riga *)
IF (CmdStart AND RicStsRun)= true THEN
	StsRun:= true;
	Index:= 1;
	CmdStart:= false;
	StsEnd:= false;
	FlagStsEnd:= false;
ELSIF RicStsRun=FALSE THEN
	StsRun:= false;
	Index:= 0;
END_IF;

FOR i:=0 TO 5 DO
	IF Index=i THEN	
		StepCiclo[i]:= true;
	ELSE
		StepCiclo[i]:= false;
	END_if;
END_FOR;

(* Cicli in base a codice azione *)
(* RIempimento acqua *)
IF RicAzione=5 THEN
	(* Passaggio parametri *)
	IF StepCiclo[1]=true THEN
		TemperaturaAcquaPerBCD:= INT_TO_WORD(((WORD_TO_INT(RicGradi)) * 10));
		LitriAcqua:= INT_TO_BCD_WORD(REAL_TO_INT(RicPeso/10,0));
		(*Controllo se è già stato eseguito un riempimento in precedenza*)
		IF FlagRiempimentoAcqua = TRUE THEN
			(*Riempimento già eseguito, richiedo la presenza operatore*)
			PopupMancatoScolaggio:= TRUE;
			IF PopupMancatoScolaggio=TRUE AND ConfermaMancatoScolaggio THEN (*Quando viene confermato il riempimento nonostante non ho scolaggio*)
				PopupMancatoScolaggio:= false;
				ConfermaMancatoScolaggio:= false;
				Index:= 2;
			END_IF;
		ELSE (*Se non è già avvenuto, proseguo*)		
			Index:= 2;
		end_if;
	END_IF;
	(*Comando*)
	IF StepCiclo[2]=true THEN
		CmdAcqua:= true;
		Index:= 3;
	END_IF;
	(* Attesa ritorno *)
	IF (StepCiclo[3] AND FeedbackAcqua)=TRUE  THEN
		FlagRiempimentoAcqua:= TRUE;
		Index:= 4;
	END_IF;
	(* Attesa fine operazione *)
	IF StepCiclo[4]=true AND FeedbackAcqua=false THEN
		TemperaturaMacchina:= TemperaturaAcqua;
		VelocBotte:= 9;
		CmdTemperaturaON:= true;
		CmdRotAv:= true;
		IF FeedbackRotAv=TRUE then
			CmdRotAv:= FALSE;
			StsRun:= false;
			StsEnd:= true;
		end_if;
	END_IF;
END_IF;

(* RIempimento formico *)
IF RicAzione=6 THEN
	(* Passaggio parametri *)
	TIMX(StepCiclo[1]=true,TimerFormico1,20);
	TIMX(StepCiclo[1]=true,TimerFormico2,40);
	TIMX(StepCiclo[2]=true,TimerFormico3,20);
	TIMX(StepCiclo[2]=true,TimerFormico4,40);
	TIMX(StepCiclo[3]=true,TimerFormico5,20);
	TIMX(StepCiclo[3]=true,TimerFormico6,40);
	IF StepCiclo[1]=true THEN
		PesoFormico:=  INT_TO_BCD_WORD(REAL_TO_INT(RicPeso*10,0));
		RichiestaFormico:= true;
		IF TimerFormico1.CF=TRUE THEN
			RichiestaFormico:= false;
			IF TimerFormico2.CF=TRUE THEN
				Index:= 2;
			END_IF;
		END_IF;
	END_IF;
	(*Comando*)
	IF StepCiclo[2]=true THEN
		SceltaFormico:= true;
		IF TimerFormico3.CF=TRUE THEN
			SceltaFormico:= false;
			IF TimerFormico4.CF=TRUE THEN
			Index:= 3;
			END_IF;
		END_IF;
	END_IF;
	(* Attesa ritorno *)
	IF StepCiclo[3] =true THEN
		CmdFormico:= true;
		IF TimerFormico5.CF=TRUE THEN
			CmdFormico:= false;
			IF TimerFormico6.CF=TRUE AND FeedbackFormico=TRUE THEN
				AutPoupupAcido:= true;
				Index:= 4;
			END_IF;
				END_IF;
	END_IF;
	(* Attesa fine operazione *)
	IF StepCiclo[4]=true AND AutPoupupAcido=false AND FeedbackFormico=false THEN
		VaiAInvioInBotte:= TRUE;
		StsRun:= false;
		StsEnd:= true;
	END_IF;
END_IF;

(* RIempimento glutaraldeide *)
IF RicAzione=7 THEN
	(* Passaggio parametri *)
	TIMX(StepCiclo[1]=true,TimerGlutar1,20);
	TIMX(StepCiclo[1]=true,TimerGlutar2,40);
	TIMX(StepCiclo[2]=true,TimerGlutar3,20);
	TIMX(StepCiclo[2]=true,TimerGlutar4,40);
	TIMX(StepCiclo[3]=true,TimerGlutar5,20);
	TIMX(StepCiclo[3]=true,TimerGlutar6,40);
	IF StepCiclo[1]=true THEN
		PesoGlutaral:=  INT_TO_BCD_WORD(REAL_TO_INT(RicPeso*10,0));
		SceltaGlutar:= true;
		IF TimerGlutar1.CF=TRUE THEN
			SceltaGlutar:= false;
			IF TimerGlutar2.CF=TRUE THEN
				Index:= 2;
			END_IF;
		END_IF;
	END_IF;
	(*Comando*)
	IF StepCiclo[2]=true THEN
		RichiestaGlutar:= true;
		IF TimerGlutar3.CF=TRUE THEN
			RichiestaGlutar:= false;
			IF TimerGlutar4.CF=TRUE THEN
			Index:= 3;
			END_IF;
		END_IF;
	END_IF;
	(* Attesa ritorno *)
	IF StepCiclo[3] =true THEN
		CmdGlutaral:= true;
		IF TimerGlutar5.CF=TRUE THEN
			CmdGlutaral:= false;
			IF TimerGlutar6.CF=TRUE AND FeedbackGlutaral=TRUE THEN
				AutPoupupAcido:= true;
				Index:= 4;
			END_IF;
				END_IF;
	END_IF;
	(* Attesa fine operazione *)
	IF StepCiclo[4]=true AND AutPoupupAcido=false AND FeedbackGlutaral=false THEN
		StsRun:= false;
		StsEnd:= true;
	END_IF;
END_IF;

(* Rotazione avanti, tipo 1 *)
IF RicAzione=10 AND RicRotaz=1 THEN
	(* Passaggio parametri *)
	IF StepCiclo[1]=true THEN
		VelocBotte:= RicSpeed;
		Index:= 2;
	END_IF;
	(*Comando*)
	IF StepCiclo[2]=true THEN
		CmdRotAv:= true;
		Index:= 3;
	END_IF;
	(* Attesa ritorno *)
	IF StepCiclo[3]=true AND FeedbackRotAv=true THEN
		TIMX(StepCiclo[3]=true,TimerRotazione,DelayRotazione);
		CmdRotAv:= false;
		IF TimerRotazione.CF THEN		
			Index:= 4;
		END_IF;
	END_IF;
	(* Attesa fine operazione *)
	IF StepCiclo[4]=true  THEN	
		StsRun:= false;
		StsEnd:= true;
	END_IF;
END_IF;

(* Rotazione indietro, tipo 2 *)
IF RicAzione=10 AND RicRotaz=2 THEN
	(* Passaggio parametri *)
	IF StepCiclo[1]=true THEN
		VelocBotte:= RicSpeed;
		Index:= 2;
	END_IF;
	(*Comando*)
	IF StepCiclo[2]=true THEN
		CmdRotInd:= true;
		Index:= 3;
	END_IF;
	(* Attesa ritorno *)
	IF StepCiclo[3]=true AND FeedbackRotInd=true THEN
		TIMX(StepCiclo[3]=true,TimerRotazione,DelayRotazione);
		CmdRotInd:= false;
		IF TimerRotazione.CF THEN		
			Index:= 4;
		END_IF;
	END_IF;
	(* Attesa fine operazione *)
	IF StepCiclo[4]=true  THEN	
		StsRun:= false;
		StsEnd:= true;
	END_IF;
END_IF;

(* Rotazione alternata, tipo 3 *)
IF RicAzione=10 AND RicRotaz=3 THEN
	(* Passaggio parametri *)
	IF StepCiclo[1]=true THEN
		VelocBotte:= RicSpeed;
		IF RicMinuti<=60 then
			DelayRotazione:= (WORD_TO_UINT(RicMinuti)*600);
			TimxTempDelay:= 0;
		ELSIF RicMinuti>60 THEN
			TimxTempDelay:= 0;
			TimxRicMinuti:= WORD_TO_INT(RicMinuti);
			WHILE TimxRicMinuti>60 DO
				TimxRicMinuti:= TimxRicMinuti-60;
				TimxTempDelay:= TimxTempDelay+1;
			END_WHILE;
			DelayRotazione:= (INT_TO_UINT(TimxRicMinuti))*600;
		end_if;
		Index:= 2;
		CmdRotAlt:= true;
	END_IF;
	(*Comando*)
	IF StepCiclo[2]=true THEN
		
		Index:= 3;
	END_IF;
	(* Attesa ritorno *)
	IF TimxTempDelay= 0 then
		TIMX(StepCiclo[3]=true,TimerRotazione3,DelayRotazione);
	ELSIF TimxTempDelay>0 THEN
		TIMX(StepCiclo[3]=true,TimerRotazione3,36000);
	end_if;
	IF StepCiclo[3]=true AND FeedbackRotAlt=true THEN
		CmdRotAlt:= false;
		IF TimerRotazione3.CF THEN
				IF TimxTempDelay= 0 then
					Index:= 4;
				ELSIF TimxTempDelay>0 THEN
					TimxTempDelay:=TimxTempDelay-1;
					Index:= 2;
				end_if;
		END_IF;
	END_IF;
	(* Attesa fine operazione *)
	IF StepCiclo[4]=true  THEN	
		StsRun:= false;
		StsEnd:= true;
	END_IF;
END_IF;

(* Ferma rotazione, tipo 4 *)
IF RicAzione=10 AND RicRotaz=4 THEN
	(* Passaggio parametri *)
	IF StepCiclo[1]=true THEN
		Index:= 2;
	END_IF;
	(*Comando*)
	IF StepCiclo[2]=true THEN
		CmdRotStop:= true;
		Index:= 3;
	END_IF;
	(* Attesa ritorno *)
	TIMX(StepCiclo[3]=true,TimerRotazione4,100);
	IF StepCiclo[3]=true THEN
		IF TimerRotazione4.CF THEN		
			CmdRotStop:= FALSE;
			Index:= 4;
		END_IF;
	END_IF;
	(* Attesa fine operazione *)
	IF StepCiclo[4]=true  THEN	
		StsRun:= false;
		StsEnd:= true;
	END_IF;
END_IF;

(* Rotazione alternata notte, tipo 5 *)
IF RicAzione=10 AND RicRotaz=5 THEN
	(* Passaggio parametri *)
	IF StepCiclo[1]=true THEN
		PopupRotNotte:= false;
		VelocBotte:= 6;
		OreAltPreNotte:= 0;
		MinAltPreNotte:= 5;
		Index:= 2;
	END_IF;
	(*Comando*)
	IF StepCiclo[2]=true THEN
		AutCmdNotturno:= TRUE;
		Index:= 3;
	END_IF;
	(* Attesa ritorno *)
	IF StepCiclo[3]=true AND FeedbackRotAlt=true THEN
			PopupRotNotte:= true;
			Index:= 4;
		END_IF;
	END_IF;
	(* Attesa fine operazione *)
	IF StepCiclo[4]=true AND ConfermaRotNotte=true  THEN
		PopupRotNotte:= false;
		StsRun:= false;
		StsEnd:= true;
	END_IF;

(* Rotazione alternata, tipo 7 *)
IF RicAzione=10 AND RicRotaz=7 THEN
	(* Passaggio parametri *)
	IF StepCiclo[1]=true THEN
		VelocBotte:= RicSpeed;
		IF RicMinuti<=60 then
			DelayRotazione:= (WORD_TO_UINT(RicMinuti)*600);
			TimxBedinaDelay:= 0;
		ELSIF RicMinuti>60 THEN
			TimxBedinaDelay:= 0;
			TimxRicMinuti:= WORD_TO_INT(RicMinuti);
			WHILE TimxRicMinuti>60 DO
				TimxRicMinuti:= TimxRicMinuti-60;
				TimxBedinaDelay:= TimxBedinaDelay+1;
			END_WHILE;
			DelayRotazione:= (INT_TO_UINT(TimxRicMinuti))*600;
		end_if;
		Index:= 2;
		CmdRotAlt:= true;
		BedinaRunning:= true;
	END_IF;
	(*Comando*)
	IF StepCiclo[2]=true THEN
		Index:= 3;
	END_IF;
	
	IF StepCiclo[3]=true AND FeedbackRotAlt=true THEN
		CmdRotAlt:= false;
	    Index:= 4;
	END_IF;
	(* Attesa fine operazione *)
	IF StepCiclo[4]=true  THEN	
		StsRun:= false;
		StsEnd:= true;
	END_IF;
END_IF;

(* Preparazione bedina, tipo 7  *)
IF RicAzione=50 AND RicRotaz=7 THEN
	(* Passaggio parametri *)
	IF StepCiclo[1]=true THEN
		VaiAInvioInBotte:= TRUE;
		RichiestaLetturaBarcode:= TRUE;
		AutPoupupBedina:= 1;
		FlagAbilitaScansioni:= TRUE;
	        	
				FlagScansioniFallite:= FALSE;
				FlagIgnoraScansioniFallite:= FALSE;
				NumeroScansioni:= 0;
				FlagRitentaScansioni:= FALSE;
				StatoScansione:= 0;
		Index:= 2;
	END_IF;
	(*Comando*)
	IF StepCiclo[2]=true AND ((LetturaPesoREAL=0,0) AND LetturaCodPro=0 AND LetturaRicetta=0) THEN
		ProdottoErratoPopup:= false;
		StatoScansione:= 1;
		Index:= 3;
	END_IF;
	(* Attesa ritorno *)

	IF StepCiclo[3]=true AND (FlagScansioniFallite=FALSE) AND (LetturaPesoREAL<>0,0) AND (LetturaCodPro<>0) AND (LetturaRicetta<>0) THEN
		(*Conversione peso da DINT da bilanca a reale, in Kg. Calcolo tolleranze da parametro tolleranza % (5%, per ora)*)
		LetturaPesoREAL:= DINT_TO_REAL(LetturaPesoDINT);
		LetturaPesoREAL:= LetturaPesoREAL/REAL1000;
		TolleranzaInf:= PesoNecessarioRicetta-((PesoNecessarioRicetta*Tolleranza)/PercentualeREAL);
		TolleranzaSup:= PesoNecessarioRicetta+((PesoNecessarioRicetta*Tolleranza)/PercentualeREAL);
		(*Su codice a barre Anno e n°Ricetta sono un codice unico, vengono uniti in quanto separati*)
		TempAnnoNecessario:= INT_TO_DINT(AnnoNecessarioRicetta);
		LetturaRicettaTemp:= (TempAnnoNecessario*10000000)+(RicettaNecessariaRicetta);
		
						
		(*Controlla corrispondeza peso, codice prodotto, codice ricetta*)
			IF LetturaPesoREAL>TolleranzaInf AND LetturaPesoREAL<TolleranzaSup AND LetturaCodPro= CodiceNecessarioRicetta AND LetturaRicetta=LetturaRicettaTemp then		
				Index:= 4;
				FlagNuovaScansione:= false;
				RichiestaLetturaBarcode:= FALSE;
				AutPoupupBedina:= 0;
				FlagAbilitaScansioni:= FALSE;
				NumeroScansioni:= 0;
				ELSE
				(*Se il prodotto non è giusto, segno 1 tentativo e resetto tutto*)
				StatoScansione:= 2;
				
				IF NumeroScansioni<2 THEN
					NumeroScansioni:= NumeroScansioni+1;
					Index:= 2;
				
				ELSIF NumeroScansioni>=2 THEN
					FlagScansioniFallite:= TRUE;
									
				END_IF;;
		
		FlagNascondiTasti:= NOT(FlagScansioniFallite OR RichiestaLetturaBarcode);
	END_IF;
				
END_IF;		
	(* Attesa fine operazione *)
		IF StepCiclo[3]=true AND FlagScansioniFallite=TRUE THEN
			IF FlagIgnoraScansioniFallite=TRUE THEN
				FlagScansioniFallite:= FALSE;
				FlagIgnoraScansioniFallite:= FALSE;
				RichiestaLetturaBarcode:= FALSE;
			    AutPoupupBedina:= 0;
				NumeroScansioni:= 0;
				Index:= 4;
			END_IF;
		END_IF;		
	(*invio in bedina manuale completato, conferma da operatore*)
	IF StepCiclo[4]=true  THEN
		
		ConfermaBedina:= False;
		RichiestaConfermaBedina:= false;
		StsRun:= false;
		StsEnd:= true;
				
	END_IF;
END_IF;

(* Invio in botte, tipo 8 *)
IF RicAzione=10 AND RicRotaz=8 THEN
	IF StepCiclo[1]=true AND BedinaTimeEnd=FALSE THEN
	AutPoupupTBedina:= 1;
	END_IF;
	(* Passaggio parametri *)
	IF StepCiclo[1]=true AND BedinaTimeEnd=TRUE THEN
		IF FlagSolido=TRUE THEN
			CmdRotStop:= true;
		end_if;
		Index:= 2;
		AutPoupupTBedina:= 0;
		BedinaTimeEnd:= FALSE;
	END_IF;
	(*Comando*)
	TIMX(StepCiclo[2]=true,TimerRotazione4,100);
	IF StepCiclo[2]=true THEN
		IF FlagSolido=TRUE THEN
			IF TimerRotazione4.CF THEN		
				CmdRotStop:= FALSE;
				Index:= 3;
				FlagSolido:= false;
				VaiAInvioInBotte:= true;
			END_IF;
		ELSE
			Index:= 3;
			VaiAInvioInBotte:= true;
		end_if;
	END_IF;
	(* Attesa ritorno *)
	IF StepCiclo[3]=true THEN
		AutPupupInvioBotte:= true;
			Index:= 4;
		(*END_IF;*)
	END_IF;
	(* Attesa fine operazione *)
	IF StepCiclo[4]=true AND ConfermaInvioBotte=true THEN	
		ConfermaInvioBotte:= false;
		AutPupupInvioBotte:= false;
		StsRun:= false;
		StsEnd:= true;
	END_IF;
END_IF;

(* Controllo *)
IF RicAzione=15 THEN
	(* Passaggio parametri *)
	IF StepCiclo[1]=true THEN
		Index:= 2;
	END_IF;
	(*Comando*)
	IF StepCiclo[2]=true THEN
		Index:= 3;
	END_IF;
	(* Attesa ritorno *)
	IF StepCiclo[3]=true THEN
		Index:= 4;
	END_IF;
	(* Attesa fine operazione *)
	IF StepCiclo[4]=true AND ConfermaControllo=True THEN	
		ConfermaControllo:= false;
		StsRun:= false;
		StsEnd:= true;
	END_IF;
END_IF;

(*Scolaggio a decremento da asse*)
IF RicScola=2 AND RicAzione= 0 THEN
	IF StepCiclo[1]=TRUE THEN
		CmdScolaggioDecrementoAsse:= true;
		IF StsScolaggioDecrementoAsse=TRUE THEN
			CmdScolaggioDecrementoAsse:= false;
			Index:= 2;
		END_IF;
	END_IF;
	IF StepCiclo[2]=TRUE THEN
		IF AutCmdStop=TRUE THEN
			FlagRiempimentoAcqua:= false;
			StsRun:= false;
			StsEnd:= true;
		END_IF;
	END_IF;
(*ELSIF RicScola=1 AND RicAzione= 0 THEN
	IF StepCiclo[1]=TRUE THEN
		CmdScolaggioNormale:= true;
		TIMX(StepCiclo[1],TimerScolaggioON,10);
		IF TimerScolaggioON.CF=TRUE THEN
			CmdScolaggioNormale:= false;
			Index:= 2;
		END_IF;
	END_IF;
	IF StepCiclo[2]=TRUE THEN
		IF StsScolaggioNormale=FALSE THEN
			StsRun:= false;
			StsEnd:= true;
		END_IF;
	END_IF;*)
IF RicScola<>0 OR RicAzione=99 then
	CmdTemperaturaOFF:= true;
	TemperaturaMacchina:= 1;
end_if;
END_IF;		
(*Con la pausa non incremento il passo a fine azione*)
IF (NOT RicPause) AND RicStart then
	(* Cambio riga su fronte dello status end. Aumenta il puntatore e carica il passo successivo*)
	IF StsEnd<>FlagStsEnd THEN
		RicStato:=2;
		PassoPuntatoreINT:= WORD_TO_INT(PassoPuntatore);
		PassoPuntatoreINT:= (PassoPuntatoreINT+1);
		PassoPuntatore:= INT_TO_WORD(PassoPuntatoreINT);
		CaricaRIcetta:= true;
	END_IF;
	FlagStsEnd:= StsEnd;
ELSE
	StsRun:= false;
END_IF;

	
(*Copia  stsRun e comandi torretta luminosa in variabili globali*)
GlobalStsRun:= StsRun;
(*Se sono in marcia automatica, controllo torretta e stati in automatico, altrimenti sono esclusi*)
IF StsRun=TRUE then
	IF RicAzione=50 OR RicAzione=10 OR RicAzione=15 then
		CASE WORD_TO_INT(RicRotaz) OF
			1..6: (*Con rotazioni standard, luce fissa*)
				GlobalGreenLight:= true;
			7: (*Se invio in bedina o in botte, la luce lampeggia*)
				GlobalGreenFlash:= true;
		END_CASE;
	END_IF;
	(*Lampeggio torretta con conferma di mancato scolaggio*)
	IF (RicAzione=5 AND PopupMancatoScolaggio=TRUE) OR (RicAzione=10 AND  RicRotaz=8 AND BedinaRunning=FALSE) OR (RicAzione=15) OR (RicAzione=6) THEN
		GlobalGreenFlash:= TRUE;
	END_IF;
    IF (RicAzione=10 AND  RicRotaz=8 AND BedinaRunning=TRUE) OR (RicAzione=0 AND RicScola=2 AND PopupMancatoScolaggio=false) THEN
		GlobalGreenLight:= TRUE;
	END_IF;
ELSE
	(*Lo StsRun si reinizializza su ogni passo, attenzione alle memorie che vengono inserite di seguito*)
	(*Resetta memoria usate dalla ricetta*)
	GlobalGreenLight:= false;
	GlobalGreenFlash:= false;
	RicAzione:= 0;
	RicRotaz:= 0;
	VisibilitàIndietroMan:= true;
	FlagRiempimentoAcqua:= false;
	CmdRotAv:= false;
	CmdRotInd:= false;
	CmdRotAlt:= false;
	IF stopDaBarriera = FALSE THEN
		CmdRotStop:= false;
	end_if;
	CmdRotNotte:= false;
	CmdAcqua:= false;
	CmdFormico:= false;
	CmdGlutaral:= false;
	CmdScolaggioDecrementoAsse:= false;
	CmdScolaggioNormale:= false;
	PopupMancatoScolaggio:= false;
	RichiestaLetturaBarcode:= false;
	AutCmdNotturno:= false;
	AutPupupInvioBotte:= false;
	AutPoupupBedina:= 0;
	AutPoupupTBedina:= 0;
	PopupRotNotte:= false;
	
	ConfermaInvioBotte:= false;
	AutPupupInvioBotte:= false;
	AutFlagConforme:= false;
END_IF;
IF rRicStsRun= FALSE AND NOT stopDaBarriera THEN
	GlobalGreenLight:= false;
	GlobalGreenFlash:= false;
	RicAzione:= 0;
	RicRotaz:= 0;
	VisibilitàIndietroMan:= true;
	FlagRiempimentoAcqua:= false;
	CmdRotAv:= false;
	CmdRotInd:= false;
	CmdRotAlt:= false;
	CmdRotStop:= false;
	CmdRotNotte:= false;
	CmdAcqua:= false;
	CmdFormico:= false;
	CmdGlutaral:= false;
	CmdScolaggioDecrementoAsse:= false;
	CmdScolaggioNormale:= false;
	PopupMancatoScolaggio:= false;
	RichiestaLetturaBarcode:= false;
	AutCmdNotturno:= false;
	AutPupupInvioBotte:= false;
	AutPoupupBedina:= 0;
	AutPoupupTBedina:= 0;
	PopupRotNotte:= false;
	
				AutPoupupTBedina:= 0;
				BedinaTimeEnd:= FALSE;
		
				FlagNuovaScansione:= false;
				RichiestaLetturaBarcode:= FALSE;
				AutPoupupBedina:= 0;
				FlagAbilitaScansioni:= FALSE;
				NumeroScansioni:= 0;
				
				ConfermaInvioBotte:= false;
				AutPupupInvioBotte:= false;
				AutFlagConforme:= false;
END_IF;
	(*Lampeggio torretta con fine ricetta*)
	IF AutRicettaENd=TRUE OR RicAzione=99 THEN
		GlobalGreenFlash:= TRUE;
	END_IF;
	
VisibilitàIndietroMan:= true;

(*(*Gestione stato della botte per supervisione*)
IF (StatoMacchina= 0) AND (PaginaAtt=2) AND RicStsRun= false THEN
	StatoMacchina:= 1;
ELSIF (PaginaAtt<>2) AND (StatoMacchina)<2 THEN
	StatoMacchina:= 0;
end_if;
IF (StatoMacchina=2 AND RicStsRun=TRUE) OR GlobalGreenLight=TRUE THEN
	StatoMacchina:= 3;
END_IF;
IF RicPause THEN
	StatoMacchina:= 4;
END_IF;
IF GlobalGreenFlash=TRUE THEN
	StatoMacchina:= 5;
END_IF;
IF RicAzione=99 THEN
	StatoMacchina:= 10;
end_if;
IF StatoMacchina=11 THEN
	StatoMacchina:= 0;
end_if;

luceProdotti:= FALSE;

IF delayAlternataOn = TRUE THEN
	CmdRotAlt := TRUE;
end_if;